///////////
// Structure For DEIECommand. Main Operating Data to be saved (ex: OPC).
//////////
TYPE GRID_Enedis :
STRUCT
	
	MesData								: GRID ; 		(* GRID MesData *)
                                       	
	OUT_CmdPReg                         : BOOL ;     	(* (NA) Passage à P0 reçu DI*)
	OUT_CmdQReg	                   	    : BOOL ;     	(* (NA) Passage à Q0 reçu DI*)

	OUT_Rse								: BOOL; 		(* (NA) Protection en Rse(1) / Protection Hors RSE (O) *)
	OUT_TA								: BOOL; 		(* (NA) Telecaction en service (1) / Teleaction Hors service (0)*)
	
END_STRUCT
END_TYPE

(* stored: Version 1.1.0.1, ProductVersion 3.1.4024.9
   DUT GRID_Enedis: Id {289c1095-8923-4439-a8ba-a8650581126f} *)
